FUNCTION_BLOCK FB_ItemBuffer
VAR_IN_OUT
	st_BufferData	:	ST_ItemBuffer;	// Buffer Type
END_VAR
VAR_INPUT
	st_BufferFdbkIn : ST_ItemBufferFdbk;	//	Buffer Feedback
END_VAR
VAR_OUTPUT
	// Output the In and Out pointer to allow testing of the 
	st_BufferFdbkOut : ST_ItemBufferFdbk;	//	Buffer Feedback
END_VAR
VAR
	nOutPointer		:	UDINT;				// OutPointer use to detect items in the buffer
	nBufferSizeTemp : 	UDINT;				// Calculate buffer size from Byte count
	nBufferSize : 	UDINT;					// Buffer Size in total elements
	st_Blank	:	ST_Item :=  (ID := '',
									UniqueID := 0,
									Destination := 0,
									Status := E_StatusCode.No_Status,
									DeviceID := '');
	nInit				: UDINT;					// Used to initialize the Array on Start-up
	nItemExtSize		: UDINT;				// Size of ST_ItemExt in Bytes
	bInitDone			: BOOL := FALSE;			// Set if Init occurred outside of FB_init
	bMaster				: BOOL := TRUE;			// Master = TRUE if this FB instance adds items to the buffer
	bLogEntries			: BOOL := FALSE;
	sBufferName			: STRING;				// Name of the Buffer for Logging Purposes
END_VAR

VAR CONSTANT
	nBITCOUNT: UINT := 32;	// Number of Bits in each Array Element
	nBYTECOUNT : UINT := 4;	// Number of Bytes in each array element
	nUDINTBYTECOUNT : UINT := 4;	// Number of Bytes in a UDINT data type
END_VAR

// This will run if FB_init did not detect a valid reference and initialize the Structure
IF NOT bInitDone THEN
(*
	// Get the Data Item In Bytes
	nBufferSizeTemp := TO_UDINT(SIZEOF(st_BufferData));
	// Reduce the byte count by the In and Out pointer byte count
	nBufferSizeTemp := nBufferSizeTemp - (nUDINTBYTECOUNT);
	// Get the size of the ST_ItemExt Data type
	nItemExtSize := TO_UDINT(SIZEOF(st_Blank));
	// Get the total number of bytes in the Array, by dividing the remaining nBufferSize by the nItemExtSize
	nBufferSize := nBufferSizeTemp/nItemExtSize;
*)
	nBufferSize := GetBufferSize();
	// Clear the buffer for the master
	// Set the OutPointer for a reader/consumer
	IF bMaster THEN
		// Clear the Buffer on Start-up because we don't know what is and is not in process
		clear();
	ELSE
		// If this is consumer, just start at the latest data point
		nOutPointer := st_BufferData.nInPointer;
	END_IF
(*
	FOR nInit := 0 TO (nBufferSize - 1) DO
		st_BufferData.aBufferData[nInit] := st_Blank;
	END_FOR 
	// Clear the Buffer In and Out pointers
	st_BufferData.nInPointer := 0;
	nOutPointer := 0;
	// Indicate that initialization occurred outside of FB_Init
	bInitDone := TRUE;
	// The master controls the buffer contents, when the buffer is clear, turn on the bClear bit
	IF bMaster THEN
		st_BufferData.bClear := TRUE;
	END_IF
	// Turn on the Buffer Empty signal regardless of Master status.
	// In system where there is no inter-plc communication, there will be no need for a non-master
	// function blocks 
	st_BufferFdbkOut.bEmpty := TRUE;
*)
	bInitDone := TRUE;
END_IF

// If this is the master and the feedback indicates that the consumer function blocks are empty
// clear the request
IF bMaster THEN
	IF st_BufferFdbkIn.bEmpty THEN
		st_BufferData.bClear := FALSE;
	END_IF
ELSE
	// If this is a consumer function block
	// Clear the buffer, even though this is all read from the master
	// the OutPointer is set to zero in the Clear method
	IF st_BufferData.bClear THEN
		Clear();
	ELSE
		st_BufferFdbkOut.bEmpty := FALSE;
	END_IF	
END_IF

METHOD PUBLIC AddItem : ST_Item
VAR_INPUT
	st_ItemToAdd	:	ST_Item;
END_VAR
// Disable the warning regarding invalid Reference from a method for IO_OUT variables
{warning disable C0371}
// Test for a Valid reference
IF __ISVALIDREF(st_BufferData) THEN
	// Increment the In Pointer using the F_CaclculateIndex
	st_BufferData.nInPointer := F_CalculateIndex(Offset := 1,InitialValue := st_BufferData.nInPointer, BufferSize := nBufferSize);
	// Add the Item to the Buffer
	st_BufferData.aBufferData[st_BufferData.nInPointer] := st_ItemToAdd;
	IF bLogEntries THEN
		logItem(bIn := TRUE
				, st_ItemToLog := st_ItemToAdd
				, nIndex := st_BufferData.nInPointer);
	END_IF
END_IF
// Restore the warning regarding invalid Reference from a method for IO_OUT variables
{warning restore C0371}
END_METHOD

PROPERTY PUBLIC BufferSize : UDINT
GET
BufferSize := nBufferSize;
END_GET
END_PROPERTY

METHOD PUBLIC Clear
VAR_INPUT
END_VAR
// Disable the warning regarding invalid Reference from a method for IO_OUT variables
{warning disable C0371}
// Test for a Valid reference
IF __ISVALIDREF(st_BufferData) THEN
	FOR nInit := 0 TO (nBufferSize - 1) DO
		st_BufferData.aBufferData[nInit] := st_Blank;
	END_FOR 
	// Clear the Buffer In and Out pointers
	st_BufferData.nInPointer := 0;
	nOutPointer := 0;
	// The master controls the buffer contents, when the buffer is clear, turn on the bClear bit
	IF bMaster THEN
		st_BufferData.bClear := TRUE;
	END_IF
	// Turn on the Buffer Empty signal regardless of Master status.
	// In system where there is no inter-plc communication, there will be no need for a non-master
	// function blocks 
	st_BufferFdbkOut.bEmpty := TRUE;
END_IF
// Restore the warning regarding invalid Reference from a method for IO_OUT variables
{warning restore C0371}
END_METHOD

METHOD FB_init : BOOL
VAR_INPUT
	bInitRetains : BOOL; // if TRUE, the retain variables are initialized (warm start / cold start)
	bInCopyCode : BOOL;  // if TRUE, the instance afterwards gets moved into the copy code (online change)
END_VAR
// ALWAYS ReInit the arrays
bInitDone := FALSE;
// Disable the warning regarding invalid Reference from a method for IO_OUT variables
{warning disable C0371}
// Test for a Valid reference
IF __ISVALIDREF(st_BufferData) THEN
(*
	// Get the Data Item In Bytes
	nBufferSizeTemp := TO_UDINT(SIZEOF(st_BufferData));
	// Reduce the byte count by the In and Out pointer byte count
	nBufferSizeTemp := nBufferSizeTemp - (nUDINTBYTECOUNT);
	// Get the size of the ST_ItemExt Data type
	nItemExtSize := TO_UDINT(SIZEOF(st_Blank));
	// Get the total number of bytes in the Array, by dividing the remaining nBufferSize by the nItemExtSize
	nBufferSize := nBufferSizeTemp/nItemExtSize;
*)
	nBufferSize := GetBufferSize();
	// Clear the Buffer on Start-up because we don't know what is and is not in process
	clear();
(*
	FOR nInit := 0 TO (nBufferSize - 1) DO
		st_BufferData.aBufferData[nInit] := st_Blank;
	END_FOR 
	// Clear the Buffer In and Out pointers
	st_BufferData.nInPointer := 0;
	nOutPointer := 0;
	// The master controls the buffer contents, when the buffer is clear, turn on the bClear bit
	IF bMaster THEN
		st_BufferData.bClear := TRUE;
	END_IF
	// Turn on the Buffer Empty signal regardless of Master status.
	// In system where there is no inter-plc communication, there will be no need for a non-master
	// function blocks 
	st_BufferFdbkOut.bEmpty := TRUE;
*)
END_IF

// Restore the warning regarding invalid Reference from a method for IO_OUT variables
{warning restore C0371}
END_METHOD

METHOD PRIVATE GetBufferSize : UDINT
VAR_INPUT
END_VAR
// Disable the warning regarding invalid Reference from a method for IO_OUT variables
{warning disable C0371}
// Test for a Valid reference
IF __ISVALIDREF(st_BufferData) THEN
	// Get the Data Item In Bytes
	nBufferSizeTemp := TO_UDINT(SIZEOF(st_BufferData));
	// Reduce the byte count by the In and Out pointer byte count
	nBufferSizeTemp := nBufferSizeTemp - (nUDINTBYTECOUNT);
	// Get the size of the ST_ItemExt Data type
	nItemExtSize := TO_UDINT(SIZEOF(st_Blank));
	// Get the total number of bytes in the Array, by dividing the remaining nBufferSize by the nItemExtSize
	nBufferSize := nBufferSizeTemp/nItemExtSize;
	GetBufferSize := nBufferSize;
END_IF

// Restore the warning regarding invalid Reference from a method for IO_OUT variables
{warning restore C0371}
END_METHOD

PROPERTY PUBLIC LogEntries : BOOL
GET
LogEntries := bLogEntries;
END_GET
SET
bLogEntries	 := LogEntries;
END_SET
END_PROPERTY

METHOD PRIVATE LogItem
VAR_INPUT
	bIn					: BOOL;
	st_ItemToLog		: ST_Item;
	nIndex				: UDINT;
END_VAR

VAR
	sTempField			: STRING;
	sTempLogData		: STRING(255);
	nStatus			: INT;
	Out_ReadString		: INT;
END_VAR
(*
	ID : STRING := '';		// Bar Code 	
	UniqueID : DINT := 0;		// Generic ID for tracking
	Destination : DINT := 0;
	Length : DINT := 0;
	Status : E_StatusCode := E_StatusCode.No_Status;
	CapturedInMetrics : BOOL;
	DeviceID:	STRING(5);	// Device ID associated with this record
	MessageType:	E_MessageIds;	// Message Type associated with this record
*)
// Prefix with the Direction 
IF bIn THEN
	sTempLogData := '>> ';
ELSE
	sTempLogData := '<< ';
END_IF

// Buffer Name
sTempField := CONCAT(sBufferName , ' ');
sTempLogData := CONCAT(sTempLogData, sTempField);

// Index
sTempField := CONCAT(UDINT_TO_STRING(nIndex), ' ');
sTempLogData := CONCAT(sTempLogData, sTempField);

// ID
sTempField := CONCAT(st_ItemToLog.ID, ' ');
sTempLogData := CONCAT(sTempLogData, sTempField);

// Unique ID
sTempField := CONCAT(DINT_TO_STRING(st_ItemToLog.UniqueID), ' ');
sTempLogData := CONCAT(sTempLogData, sTempField);

// Destination
sTempField := CONCAT(DINT_TO_STRING(st_ItemToLog.Destination), ' ');
sTempLogData := CONCAT(sTempLogData, sTempField);

// Status
nStatus := st_ItemToLog.Status;
sTempField := CONCAT(INT_TO_STRING(nStatus), ' ');
sTempLogData := CONCAT(sTempLogData, sTempField);

// DeviceID
sTempField := CONCAT(st_ItemToLog.DeviceID, ' ');
sTempLogData := CONCAT(sTempLogData, sTempField);

// MessageType
nStatus := st_ItemToLog.MessageType;
sTempLogData := CONCAT(sTempLogData, INT_TO_STRING(nStatus));

ADSLOGSTR( msgCtrlMask := ADSLOG_MSGTYPE_HINT OR ADSLOG_MSGTYPE_LOG
		, msgFmtStr := '%s'
		, strArg := sTempLogData);
END_METHOD

PROPERTY PUBLIC Master : BOOL
GET
Master := bMaster;
END_GET
SET
bMaster := Master;
END_SET
END_PROPERTY

PROPERTY PUBLIC Name : STRING
GET
Name := sBufferName;
END_GET
SET
sBufferName := Name;
END_SET
END_PROPERTY

PROPERTY PUBLIC OutPointer : UDINT
GET
OutPointer := nOutPointer;
END_GET
END_PROPERTY

METHOD PUBLIC RemoveItem : ST_Item
VAR_OUTPUT
	st_ItemToReturn	:	ST_Item;
END_VAR
// Disable the warning regarding invalid Reference from a method for IO_OUT variables
{warning disable C0371}
// Test for a Valid reference
IF __ISVALIDREF(st_BufferData) THEN
	// Allow items out of the buffer only when not being commanded to clear the buffer
	IF NOT st_BufferData.bClear THEN
		// Increment the In Pointer using the F_CaclculateIndex
		nOutPointer := F_CalculateIndex(Offset := 1,InitialValue := nOutPointer, BufferSize := nBufferSize);
		// Add the Item to the Buffer
		st_ItemToReturn := st_BufferData.aBufferData[nOutPointer];
		IF bLogEntries THEN
			logItem(bIn := FALSE
					, st_ItemToLog := st_ItemToReturn
					, nIndex := nOutPointer);
		END_IF
	END_IF
END_IF
// Restore the warning regarding invalid Reference from a method for IO_OUT variables
{warning restore C0371}
END_METHOD

END_FUNCTION_BLOCK

(* stored: Version 1.1.0.1, ProductVersion 3.1.4024.6
   POU FB_ItemBuffer: Id {b8942154-cef3-4093-8710-a07ad33b0cef}, SpecialFunc None
   Method AddItem: Id {917e7bed-0bb9-43f1-993a-bd5979c2cdc0}
   Property BufferSize: Id {d66955f3-9f49-4f19-8330-5e6e487047cd}
   Get Get: Id {a1b3ed98-69ce-4636-bebb-547412379ebd}
   Method Clear: Id {51778ba0-d78a-4262-b617-a9567c889200}
   Method FB_init: Id {a42ee925-d6a0-42c6-a732-4a94780d0a60}
   Method GetBufferSize: Id {08d15760-f938-42e6-a937-905222c4b75e}
   Property LogEntries: Id {3cfed669-eaaf-474c-a9b3-dcdc14d13313}
   Get Get: Id {7c61944d-e3ba-44d7-a5d7-ea328f9bf42f}
   Set Set: Id {eda7b105-8bb1-414e-a529-6b89fd5817c2}
   Method LogItem: Id {0bd46e52-cff5-4362-a3ba-2cd396931de3}
   Property Master: Id {3834c791-234a-495e-9a46-796affa0e843}
   Get Get: Id {17cf0c40-7825-4744-b9b5-7f38af05dad8}
   Set Set: Id {b2d9eb16-c70c-4462-8554-445088e93846}
   Property Name: Id {bf5c2c02-54db-4975-9df0-817514aa9163}
   Get Get: Id {d99369eb-f872-434e-b39e-edd6e23db12a}
   Set Set: Id {fb1e3497-c904-418b-854c-df2a1b591eec}
   Property OutPointer: Id {441edbb5-2d4b-48f8-947d-205a5ece9226}
   Get Get: Id {4e317439-bc28-475d-abe2-e7edf3f0681e}
   Method RemoveItem: Id {b25608c3-430c-4095-b642-b2f6ccbc1c7e} *)
